FUNCTION_BLOCK IntQueue EXTENDS Queue
VAR
	elements : FB_BA_DynamicArray := (uiEntrySize := SIZEOF(INT), uiMinExpCount := Consts.initArraySize);
	//length : USINT := 0;
END_VAR

METHOD clear : BOOL
VAR_INPUT
END_VAR
elements.Reset();
length := 0;
END_METHOD

METHOD contains : BOOL
VAR_INPUT
	value : INT;
END_VAR
VAR
	temp : INT;
	i : INT;
END_VAR
IF length = 0 THEN
	contains := FALSE;
	RETURN;
END_IF

FOR i:=0 TO (length-1) BY 1 DO
	temp := get(i);
	IF MEMCMP(ADR(temp), ADR(value), SIZEOF(INT)) = 0 THEN
		contains := TRUE;
		RETURN;
	END_IF
END_FOR
contains := FALSE;
END_METHOD

METHOD get : INT
VAR_INPUT
	i : INT;
END_VAR
elements.GetEntry(diIndex := i, pResultEntry := ADR(get));
END_METHOD

METHOD isEmpty : BOOL
VAR_INPUT
END_VAR
isEmpty := (elements.diCount = 0);
END_METHOD

METHOD poll : INT
VAR_INST
	temp : INT;
	i : UINT;
END_VAR
temp := get(i := 0);
elements.RemoveEntry(diIndex := 0);
//length := length - 1;
poll := temp;
END_METHOD

METHOD push : BOOL
VAR_INPUT
	value : INT;
END_VAR
elements.AddEntry(pEntry := ADR(value));
//length := length + 1;
END_METHOD

METHOD set : BOOL
VAR_INPUT
	i : INT;
	value : INT;
END_VAR
IF i > 0 AND i < length THEN
	elements.SetEntry(i, ADR(value));
	set := TRUE;
END_IF
END_METHOD

METHOD size : DINT
VAR_INPUT
END_VAR
size := elements.diCount;
END_METHOD

END_FUNCTION_BLOCK

(* stored: Version 1.1.0.1, ProductVersion 3.1.4024.11
   POU IntQueue: Id {b88eabe4-fa96-488a-9c59-79d0926b2421}, SpecialFunc None
   Method clear: Id {efa9c721-572f-404c-8da7-db02b1e1c076}
   Method contains: Id {fa3f73b0-bcc5-4e66-a9fa-92a1749db9fc}
   Method get: Id {f77f5f86-6803-4a8e-a82e-15512b7a2d13}
   Method isEmpty: Id {2e909f5b-f462-464b-a4f4-530341b5a502}
   Method poll: Id {d7ffe0bd-a70d-474f-b52b-bb90a8761c71}
   Method push: Id {4f38a899-fe5c-4539-b0ae-ab2eb4fd4d3f}
   Method set: Id {5fc725fe-0703-463b-b796-422a25b4ff1f}
   Method size: Id {af0b9551-be39-498e-a520-c313ac29b4d9} *)
